GLOBALCONSTANTS IG5_Device_Classes (* Industry Group 5 specific device classes (vehicle systems) *)
  (* Standard: 61499-1 *)
  (* Version 1.0, 2026-06-30, Franz Höpfinger, Demmler Andreas Fahrzeugbau *)
  PACKAGE isobus::pgn::const;
  VAR_GLOBAL CONSTANT
    DC_INDUSTRIAL_GEN_SET : BYTE := 0; (* Device Class / Vehicle System: Industrial-Process Control-Stationary (Gen-Sets) *)
    DC_NOT_AVAILABLE : BYTE := 127; (* Device Class / Vehicle System: Not Available *)
  END_VAR
END_GLOBALCONSTANTS
